SUBAPPLICATION AX_SoftkeyToggle_TO_QXA_BG (* Softkey (Key-Release) kippt ein Toggle-Flip-Flop (AX_T_FF) auf QXA, Background spiegelt den Zustand. Generisch. *)
  (* Standard: 61499-2 *)
  (* Version 1.0, 2026-09-09, Franz Höpfinger, Meisterschulen am Ostbahnhof, Ausgelagert aus Uebung_010d2_sub_AX zur Wiederverwendung; u16ObjId/Output zuvor fest importiert (SoftKey_F1/Output_Q1), jetzt generische Defaults (ID_NULL/Invalid). *)
  PACKAGE MyLib::sys;
  IMPORT isobus::UT::Q::const::IDs::ID_NULL;
  IMPORT logiBUS::io::DQ::logiBUS_DO;
  IMPORT logiBUS::io::DQ::logiBUS_DO_S;
  IMPORT isobus::UT::io::Softkey::SoftKeyActivationCode::SK_RELEASED;
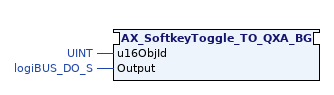
  VAR_INPUT
    u16ObjId : UINT := ID_NULL; (* Object ID *)
    Output : logiBUS::io::DQ::logiBUS_DO_S := logiBUS_DO::Invalid; (* Identify the Output Output_Q1..Q8 *)
  END_VAR
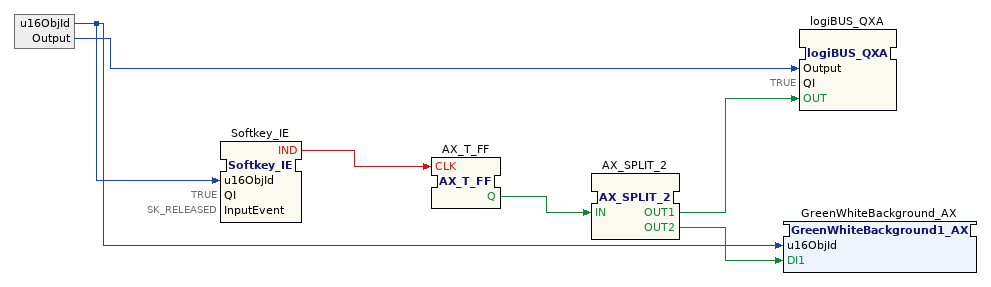
  FBS
    Softkey_IE : isobus::UT::io::Softkey::Softkey_IE(QI := TRUE, InputEvent := SK_RELEASED);
    AX_T_FF : adapter::events::unidirectional::AX_T_FF;
    AX_SPLIT_2 : adapter::events::unidirectional::AX_SPLIT_2;
    logiBUS_QXA : logiBUS::io::DQ::logiBUS_QXA(QI := TRUE);
  END_FBS
  SUBAPPS
    GreenWhiteBackground_AX : MyLib::sys::GreenWhiteBackground1_AX;
  END_SUBAPPS
  EVENT_CONNECTIONS
    Softkey_IE.IND TO AX_T_FF.CLK;
  END_CONNECTIONS
  DATA_CONNECTIONS
    u16ObjId TO Softkey_IE.u16ObjId;
    u16ObjId TO GreenWhiteBackground_AX.u16ObjId;
    Output TO logiBUS_QXA.Output;
  END_CONNECTIONS
  ADAPTER_CONNECTIONS
    AX_T_FF.Q TO AX_SPLIT_2.IN;
    AX_SPLIT_2.OUT1 TO logiBUS_QXA.OUT;
    AX_SPLIT_2.OUT2 TO GreenWhiteBackground_AX.DI1;
  END_CONNECTIONS
END_SUBAPPLICATION
